// TIA Portal V17 export
// export: Created 2025-06-26T07:49:56.9863004Z, ExportSetting WithDefaults, DisplayName Totally Integrated Automation Portal, DisplayVersion V17 Update 8, DisplayName TIA Portal Openness, DisplayVersion V17 Update 8, DisplayName TIA Portal Version Control Interface, DisplayVersion V17, DisplayName STEP 7 Professional, DisplayVersion V17 Update 8, DisplayName STEP 7 Safety, DisplayVersion V17 Update 6, DisplayName WinCC Advanced, DisplayVersion V17 Update 8
TYPE "stTrackingRegulator"
// stored: IsFailsafeCompliant false
   STRUCT
      bEnable : Bool;   // 1 = controller enabled, 0 = disabled
      fSP : Real;   // Setpoint (eg °C)
      fPV : Real;   // Process value (eg °C)
      fPVvelocity : Real;   // Rate of change of process value (eg °C/sec)
      fOutMax : Real;   // Positive-most manipulated value (eg %)
      fOutMin : Real;   // Negative-most manipulated value (eg %)
      fOut : Real;   // Manipulated value (eg %)
      bManualMode : Bool;   // 1 = manual mode, 0 = auto
      fManualValue : Real;   // Fixed manipulated value (eg %)
      fSlewRatePositive : Real;   // Controller ramp in positive direction (eg %/s)
      fSlewRateNegative : Real;   // Controller ramp in negative direction (eg %/s)
      fHysteresis : Real;   // Deadband around setpoint (eg °C)
      fVelocityPositiveLimit : Real;   // Max positive rate of change of process value (eg °C/s)
      fVelocityNegativeLimit : Real;   // Max negative rate of change of process value (eg °C/s)
      bAtMin : Bool;   // Controller negative saturation
      bAtMax : Bool;   // Controller positive saturation
      bAtSetpoint : Bool;   // Controller within control deadband
      bFault : Bool;   // 1 = controller fault, 0 = ok
      nMode : USInt;   // 0 = Off, 1 = Auto, 2 = Manual
   END_STRUCT;
END_TYPE
